{attribute 'GeneratedUsingTerminal: IODEVICETYPE_ETHERCATPROT'}
{attribute addProperty BoxType "IODEVICETYPE_ETHERCATPROT"}
{attribute addProperty Id "Beckhoff_EPP1xxxBeckhoff_EPP1xxx_EA0FD067682Beckhoff_EPP2xxxBeckhoff_EPP2xxx_CC9FFF9D1956Beckhoff_EPP3xxxBeckhoff_EPP3xxx_6AF206961280Beckhoff_EPP4xxxBeckhoff_EPP4xxx_F9671039166Beckhoff_EPP5xxxBeckhoff_EPP5xxx_BBCFF56C232Beckhoff_EPP6xxxBeckhoff_EPP6xxx_EBEB3520594Beckhoff_EPP7xxxBeckhoff_EPP7xxx_68E6213C478Beckhoff_EPP9xxxBeckhoff_EPP9xxx_2BBF558F86SyncUnitsSyncUnits_99E584AF18InputsInputs_25A0042B160OutputsOutputs_2397A10E106InfoDataInfoData_C76BEFB322"}
{attribute addProperty CRC "2711242638"}
{attribute addProperty Size "5780"}
TYPE EtherCAT_Master_EPPxxxx_A19A478E :
STRUCT
	{attribute addProperty Name "Beckhoff_EPP1xxx"}
	{attribute addProperty PreviousPort "EtherCAT_Master_EPPxxxx : Master"}
	Beckhoff_EPP1xxx : Beckhoff_EPP1xxx_EA0FD067;
	{attribute addProperty Name "Beckhoff_EPP2xxx"}
	{attribute addProperty PreviousPort "Beckhoff EPP1xxx : C"}
	Beckhoff_EPP2xxx : Beckhoff_EPP2xxx_CC9FFF9D;
	{attribute addProperty Name "Beckhoff_EPP3xxx"}
	{attribute addProperty PreviousPort "Beckhoff EPP2xxx : C"}
	Beckhoff_EPP3xxx : Beckhoff_EPP3xxx_6AF20696;
	{attribute addProperty Name "Beckhoff_EPP4xxx"}
	{attribute addProperty PreviousPort "Beckhoff EPP3xxx : C"}
	Beckhoff_EPP4xxx : Beckhoff_EPP4xxx_F9671039;
	{attribute addProperty Name "Beckhoff_EPP5xxx"}
	{attribute addProperty PreviousPort "Beckhoff EPP4xxx : C"}
	Beckhoff_EPP5xxx : Beckhoff_EPP5xxx_BBCFF56C;
	{attribute addProperty Name "Beckhoff_EPP6xxx"}
	{attribute addProperty PreviousPort "Beckhoff EPP5xxx : C"}
	Beckhoff_EPP6xxx : Beckhoff_EPP6xxx_EBEB3520;
	{attribute addProperty Name "Beckhoff_EPP7xxx"}
	{attribute addProperty PreviousPort "Beckhoff EPP6xxx : C"}
	Beckhoff_EPP7xxx : Beckhoff_EPP7xxx_68E6213C;
	{attribute addProperty Name "Beckhoff_EPP9xxx"}
	{attribute addProperty PreviousPort "Beckhoff EPP7xxx : C"}
	Beckhoff_EPP9xxx : Beckhoff_EPP9xxx_2BBF558F;
	{attribute addProperty Name "SyncUnits"}
	SyncUnits : SyncUnits_99E584AF;
	{attribute addProperty Name "Inputs"}
	Inputs : Inputs_25A0042B;
	{attribute addProperty Name "Outputs"}
	Outputs : Outputs_2397A10E;
	{attribute addProperty Name "InfoData"}
	InfoData : InfoData_C76BEFB3;
END_STRUCT
END_TYPE

(* stored: Version 1.2.0.0, ProductVersion 3.1.4024.9
   DUT EtherCAT_Master_EPPxxxx_A19A478E: Id {66f45c7e-1a98-4ec8-bd83-4cf1fbc4784c} *)
